PROGRAM Anlage
VAR
	UR5				:FB_Roboter;
	Gripper			:FB_SmartGripper;
END_VAR

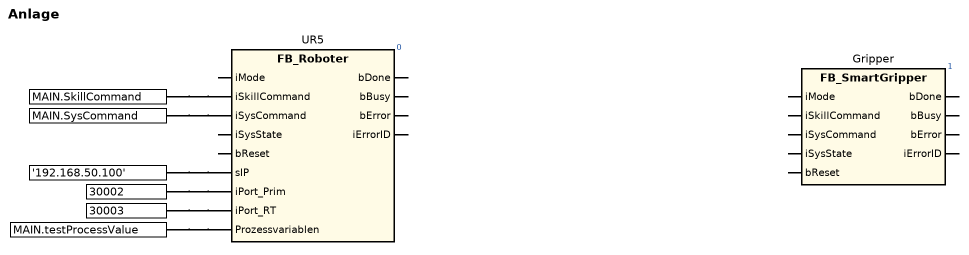
UR5(
    iSkillCommand := MAIN.SkillCommand,
    iSysCommand := MAIN.SysCommand,
    sIP := '192.168.50.100',
    iPort_Prim := 30002,
    iPort_RT := 30003,
    Prozessvariablen := MAIN.testProcessValue); // FB_Roboter
Gripper(); // FB_SmartGripper

END_PROGRAM

(* stored: Version 1.1.0.1
   POU Anlage: Id {cb61ef4c-2dc6-4929-b922-044af0a6b977}, SpecialFunc None *)
